FUNCTION_BLOCK TEST_ADD2 (* Test ADD functions *)
  (* Standard: IEC 61499-1 *)
  (* Version 0.0, 2006-09-11, JHC, Holobloc Inc *)
  (* Compiler header: package fb.rt.test; *)
  (* Compiler classdef: SimpleFB *)
  (* Compiler Java Sun JDK 1.5.0 *)
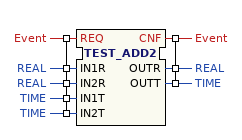
  EVENT_INPUT
    REQ WITH IN1R, IN2R, IN2T, IN1T;
  END_EVENT
  EVENT_OUTPUT
    CNF WITH OUTR, OUTT;
  END_EVENT
  VAR_INPUT
    IN1R : REAL;
    IN2R : REAL;
    IN1T : TIME;
    IN2T : TIME;
  END_VAR
  VAR_OUTPUT
    OUTR : REAL;
    OUTT : TIME;
  END_VAR
  ALGORITHM REQ IN FBD:
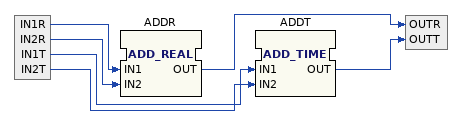
    FBS
      ADDR : ADD_REAL;
      ADDT : ADD_TIME;
    END_FBS
    DATA_CONNECTIONS
      IN1R TO ADDR.IN1;
      IN2R TO ADDR.IN2;
      ADDR.OUT TO OUTR;
      IN1T TO ADDT.IN1;
      IN2T TO ADDT.IN2;
      ADDT.OUT TO OUTT;
    END_CONNECTIONS
  END_ALGORITHM
END_FUNCTION_BLOCK
